FUNCTION TFClearWorkAreaStateSlab : BOOL
VAR_INPUT
	WorkAreaState : POINTER TO ARRAY [1..MAXAREA] OF TFMachinePalletizer_WorkAreaState;
	k : UINT;
END_VAR
VAR
	i : uINT;
	j : UINT;
END_VAR

TFClearWorkAreaStateSlab := FALSE;

FOR i:=1 TO MAXFORMINGPACK DO
	FOR j:=1 TO MAXHANDLINGSTACK DO
		WorkAreaState^[k].Slab[j] := EmptySlab;
	END_FOR
END_FOR
TFClearWorkAreaStateSlab := TRUE;

END_FUNCTION

(* stored: Version 1.1.0.1, ProductVersion 3.1.4024.11
   POU TFClearWorkAreaStateSlab: Id {da705f16-5c66-474a-9120-cc1b83f7af4c}, SpecialFunc None *)
